// TIA Portal V16 export
// export: Created 2021-09-16T19:23:48.2768921Z, ExportSetting WithDefaults, DisplayName Totally Integrated Automation Portal, DisplayVersion V16 Update 4, DisplayName TIA Portal Version Control Interface, DisplayVersion V16 Update 2, DisplayName TIA Portal Openness, DisplayVersion V16 Update 4, DisplayName STEP 7 Professional, DisplayVersion V16 Update 4, DisplayName STEP 7 Safety, DisplayVersion V16, DisplayName WinCC Advanced, DisplayVersion V16 Update 4
FUNCTION_BLOCK "Main_Safety_RTG1"   // FB1, F_FBD
{ S7_Optimized_Access := 'TRUE' }
VERSION : 0.1
// stored: AutoNumber false, IsIECCheckEnabled false, UDAEnableTagReadback false
   VAR
      faults_clear : Bool;
      last_estop_clear : Bool;
      last_reset : Bool;
   END_VAR
   VAR_TEMP   // added for the SCL form of the ladder/FBD networks
      _w1 : Bool;
      _w2 : Bool;
   END_VAR
BEGIN

REGION Network 1
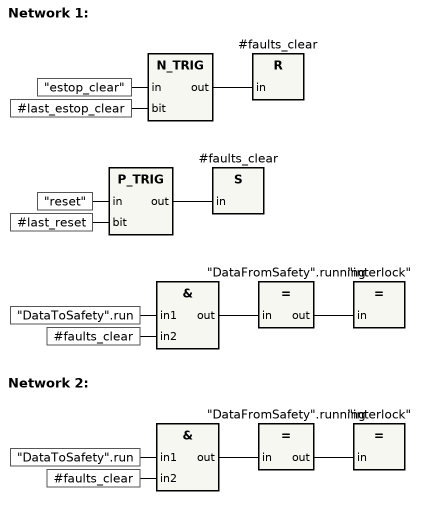
   #_w1 := NOT "estop_clear" AND #last_estop_clear;   // falling edge
   #last_estop_clear := "estop_clear";
   IF #_w1 THEN #faults_clear := FALSE; END_IF;
   #_w2 := "reset" AND NOT #last_reset;   // rising edge
   #last_reset := "reset";
   IF #_w2 THEN #faults_clear := TRUE; END_IF;
   "DataFromSafety".running := "DataToSafety".run AND #faults_clear;
   "interlock" := "DataFromSafety".running;
END_REGION

REGION Network 2
   "DataFromSafety".running := "DataToSafety".run AND #faults_clear;
   "interlock" := "DataFromSafety".running;
END_REGION
END_FUNCTION_BLOCK
